(* CoDeSys 2.3 export: FK15PUMPMANUALCONTROL.EXP *)

(* POU K15/fK15PumpManualControl, ST *)
FUNCTION fK15PumpManualControl : BOOL
VAR_INPUT
	PumpID : USINT;
	TurnOn : BOOL;
	TurnOff : BOOL;
	State : BOOL;
	EmergencyStop : BOOL;
END_VAR
VAR
END_VAR
IF TurnOn OR State THEN (*Нажата кнопка "Пуск насоса" или Работает насос?*)
	IF TurnOff THEN (*Нажата кнопка "Стоп насоса"?*)
		RETURN;
	ELSE
		IF EmergencyStop THEN (*Нажат аварийный стоп насоса?*)
			RETURN;
		ELSE
			fTurnOnK15Pump(PumpID);
		END_IF;
	END_IF;
ELSE
	RETURN;
END_IF;
END_FUNCTION
